// TIA Portal V15.1 export
// export: Created 2024-05-17T05:38:13.732926Z, ExportSetting WithDefaults, DisplayName Totally Integrated Automation Portal, DisplayVersion V15.1 Update 5, DisplayName TIA Portal Openness, DisplayVersion V15.1 Update 5, DisplayName SINAMICS Startdrive Advanced, DisplayVersion V15.1, DisplayName G130, G150, S120, S150, SINAMICS MV, S210, DisplayVersion V15.1, DisplayName G110M, G120, G120C, G120D, G120P, DisplayVersion V15.1, DisplayName STEP 7 Professional, DisplayVersion V15.1 Update 5, DisplayName STEP 7 Safety, DisplayVersion V15.1, DisplayName WinCC Professional, DisplayVersion V15.1 Update 5, DisplayName SIMATIC Visualization Architect, DisplayVersion V15.1
DATA_BLOCK "_F209000NCP01Safety"   // DB7000, F_DB
{ S7_Optimized_Access := 'TRUE' }
AUTHOR : VCC
VERSION : 0.0.0.0
// stored: AutoNumber false, DBAccessibleFromOPCUA true
   VAR
      NotUsedBool { ExternalAccessible := 'False'; ExternalVisible := 'False'; ExternalWritable := 'False'} : Bool;   // Not Used Bool
      SafetyTrue { ExternalAccessible := 'False'; ExternalVisible := 'False'; ExternalWritable := 'False'} : Bool;   // TRUE
      SafetyFalse { ExternalAccessible := 'False'; ExternalVisible := 'False'; ExternalWritable := 'False'} : Bool;   // FALSE
      HMIPassivationReset { ExternalAccessible := 'False'; ExternalVisible := 'False'; ExternalWritable := 'False'} : Bool;   // Passivation Reset from HMI
      ResetPassivation { ExternalAccessible := 'False'; ExternalVisible := 'False'; ExternalWritable := 'False'} : Bool;   // Reset Passivation
      AllSStopOk { ExternalAccessible := 'False'; ExternalVisible := 'False'; ExternalWritable := 'False'} : Bool;   // All SStop Ok
      FromPLC308_RecvError { ExternalAccessible := 'False'; ExternalVisible := 'False'; ExternalWritable := 'False'} : Bool;   // Communication Error
      FromPLC308_RecvSubsOn { ExternalAccessible := 'False'; ExternalVisible := 'False'; ExternalWritable := 'False'} : Bool;   // Outputs the fail-safe values assigned as SUBBO_xx and SUBI_xx inputs
      FromPLC308_ACK_REQ { ExternalAccessible := 'False'; ExternalVisible := 'False'; ExternalWritable := 'False'} : Bool;   // Communication Request Acknowledgement
      FromPLC308_SendMode { ExternalAccessible := 'False'; ExternalVisible := 'False'; ExternalWritable := 'False'} : Bool;   // 1=F-CPU with SENDP in deactivated safety mode
      FromPLC308_EStop_308230ZS01 { ExternalAccessible := 'False'; ExternalVisible := 'False'; ExternalWritable := 'False'} : Bool;   // PN/PN Safety Signals From external PLC
      FromPLC308_EStop_308210ZS01 { ExternalAccessible := 'False'; ExternalVisible := 'False'; ExternalWritable := 'False'} : Bool;   // PN/PN Safety Signals From external PLC
      FromPLC308_GStop_308230ZS01 { ExternalAccessible := 'False'; ExternalVisible := 'False'; ExternalWritable := 'False'} : Bool;   // PN/PN Safety Signals From external PLC
      FromPLC308_GStop_308210ZS01 { ExternalAccessible := 'False'; ExternalVisible := 'False'; ExternalWritable := 'False'} : Bool;   // PN/PN Safety Signals From external PLC
      FromPLC308_TStop_308210ZS01 { ExternalAccessible := 'False'; ExternalVisible := 'False'; ExternalWritable := 'False'} : Bool;   // PN/PN Safety Signals From external PLC
      FromPLC308_SpareBit5 { ExternalAccessible := 'False'; ExternalVisible := 'False'; ExternalWritable := 'False'} : Bool;   // PN/PN Safety Signals From external PLC
      FromPLC308_SpareBit6 { ExternalAccessible := 'False'; ExternalVisible := 'False'; ExternalWritable := 'False'} : Bool;   // PN/PN Safety Signals From external PLC
      FromPLC308_SpareBit7 { ExternalAccessible := 'False'; ExternalVisible := 'False'; ExternalWritable := 'False'} : Bool;   // PN/PN Safety Signals From external PLC
      FromPLC308_SpareBit8 { ExternalAccessible := 'False'; ExternalVisible := 'False'; ExternalWritable := 'False'} : Bool;   // PN/PN Safety Signals From external PLC
      FromPLC308_SpareBit9 { ExternalAccessible := 'False'; ExternalVisible := 'False'; ExternalWritable := 'False'} : Bool;   // PN/PN Safety Signals From external PLC
      FromPLC308_SpareBit10 { ExternalAccessible := 'False'; ExternalVisible := 'False'; ExternalWritable := 'False'} : Bool;   // PN/PN Safety Signals From external PLC
      FromPLC308_SpareBit11 { ExternalAccessible := 'False'; ExternalVisible := 'False'; ExternalWritable := 'False'} : Bool;   // PN/PN Safety Signals From external PLC
      FromPLC308_SpareBit12 { ExternalAccessible := 'False'; ExternalVisible := 'False'; ExternalWritable := 'False'} : Bool;   // PN/PN Safety Signals From external PLC
      FromPLC308_SpareBit13 { ExternalAccessible := 'False'; ExternalVisible := 'False'; ExternalWritable := 'False'} : Bool;   // PN/PN Safety Signals From external PLC
      FromPLC308_SpareBit14 { ExternalAccessible := 'False'; ExternalVisible := 'False'; ExternalWritable := 'False'} : Bool;   // PN/PN Safety Signals From external PLC
      FromPLC308_SpareBit15 { ExternalAccessible := 'False'; ExternalVisible := 'False'; ExternalWritable := 'False'} : Bool;   // PN/PN Safety Signals From external PLC
      FromPLC308_RD_I_00 { ExternalAccessible := 'False'; ExternalVisible := 'False'; ExternalWritable := 'False'} : Int;   // PN/PN Safety Signals From external PLC
      FromPLC308_RD_I_01 { ExternalAccessible := 'False'; ExternalVisible := 'False'; ExternalWritable := 'False'} : Int;   // PN/PN Safety Signals From external PLC
      ToPLC308_SendError { ExternalAccessible := 'False'; ExternalVisible := 'False'; ExternalWritable := 'False'} : Bool;   // Communication Error
      ToPLC308_SendSubsOn { ExternalAccessible := 'False'; ExternalVisible := 'False'; ExternalWritable := 'False'} : Bool;   // Outputs the fail-safe values assigned as SUBBO_xx and SUBI_xx inputs
   END_VAR
BEGIN
END_DATA_BLOCK
